// TIA Portal V18 export
DATA_BLOCK "PROFINET_NODES_WARNING"   // DB11
{ S7_Optimized_Access := 'TRUE' }
VERSION : 0.1
// stored: AutoNumber true, DBAccessibleFromOPCUA true, DBAccessibleFromWebserver true
   VAR
      AlwaysFALSE : Bool;
      AlwaysTRUE : Bool;
      "No Operation" : Bool;
      "n0010-mc1-cc1-k66001 192.168.50.10" : Bool;
      "n0010-mc2-cc1-k66001 192.168.51.10" : Bool;
   END_VAR
BEGIN
END_DATA_BLOCK
